FUNCTION_BLOCK fb_manual
VAR_INPUT
END_VAR
VAR_OUTPUT
END_VAR
VAR
	SFCInit : BOOL;
	fbi_paramInit: fb_paramInit;
	trn_paramInitDone: BOOL;

	fbi_jogController: fb_jogController;
	fbi_PTP : fb_PTP;
	fbi_operationElecylinder : fb_operationElecylinder;
	fbi_gm_operationElecylinder :fb_gm_operationElecylinder;
	fbi_oeprationChuck : fb_oeprationChuck;
	fbi_oeprationPush :fb_oeprationPush;
	fbi_operationEjector : fb_operationEjector;
	fbi_gm_operationEjector : fb_gm_operationEjector;
	fbi_recordingSystem : fb_recordingSystem;
	fbi_productGenerater : fb_productGenerator;
	fbi_gm_operationSV	: fb_gm_operationSV;
	var_i: INT;
	fbi_gm_setting: fb_gm_setting;
	fbi_gm_PTP: fb_gm_PTP;
	fbi_debugData: fb_debugData;
	var_cav_i: INT;
END_VAR

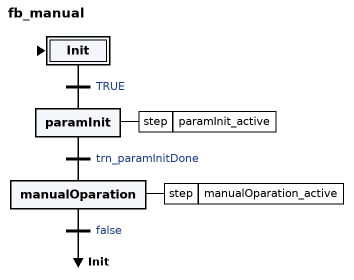
INITIAL_STEP Init:
END_STEP
TRANSITION FROM Init TO paramInit
    := TRUE;
END_TRANSITION
STEP paramInit:
    paramInit_active(N);  // step action
END_STEP
TRANSITION FROM paramInit TO manualOparation
    := trn_paramInitDone;
END_TRANSITION
STEP manualOparation:
    manualOparation_active(N);  // step action
END_STEP
TRANSITION FROM manualOparation TO Init
    := false;
END_TRANSITION

ACTION manualOparation_active:
IF manualOparation._x AND manualOparation.x = FALSE THEN
	THIS^.fbi_PTP();
	THIS^.fbi_PTP.p_init := TRUE;
	THIS^.fbi_operationElecylinder();
	THIS^.fbi_operationElecylinder.p_Init := TRUE;
	THIS^.fbi_gm_operationElecylinder();
	THIS^.fbi_gm_operationElecylinder.p_Init := TRUE;
	THIS^.fbi_oeprationChuck();
	THIS^.fbi_oeprationChuck.p_Init := TRUE;
	THIS^.fbi_oeprationPush();
	THIS^.fbi_oeprationPush.p_Init := TRUE;
	THIS^.fbi_operationEjector();
	THIS^.fbi_operationEjector.p_Init := TRUE;
	THIS^.fbi_gm_operationEjector();
	THIS^.fbi_gm_operationEjector.p_Init := TRUE;
	THIS^.fbi_gm_operationSV();
	THIS^.fbi_gm_operationSV.p_Init := TRUE;
	fbi_gm_PTP(in_flg_run := FALSE);
	//test mode
	fbi_debugData();
ELSIF manualOparation._x AND manualOparation.x THEN
	
//operation jog
	THIS^.fbi_jogController();
//PTP
	THIS^.fbi_PTP();
	THIS^.fbi_PTP.p_init := FALSE;
	fbi_gm_PTP(in_flg_run := TRUE);
//operation elecylinder
	THIS^.fbi_operationElecylinder();
	THIS^.fbi_operationElecylinder.p_Init := FALSE;
	THIS^.fbi_gm_operationElecylinder();
	THIS^.fbi_gm_operationElecylinder.p_Init := FALSE;
//operation chuck
	THIS^.fbi_oeprationChuck();
	THIS^.fbi_oeprationChuck.p_Init := FALSE;
	THIS^.fbi_gm_operationSV();
	THIS^.fbi_gm_operationSV.p_Init := FALSE;
//operation push
	THIS^.fbi_oeprationPush();
	THIS^.fbi_oeprationPush.p_Init := FALSE;
//operation ejector
	THIS^.fbi_operationEjector();
	THIS^.fbi_operationEjector.p_Init := FALSE;
	THIS^.fbi_gm_operationEjector();
	THIS^.fbi_gm_operationEjector.p_Init := FALSE;
//recording teach position
	THIS^.fbi_recordingSystem();
	fbi_gm_setting();
//new product generater
	THIS^.fbi_productGenerater();
//reset defective qty
	IF gvl_visu.flg_btn_clrDefectiveQty THEN
		FOR var_i := 1 TO 8 BY 1 DO
			gvl_auto.var_defectiveLens[var_i] := 0;
		END_FOR
	END_IF
//reset pocket qty
	IF gvl_visu.flg_btn_clrPockertQty THEN
		gvl_auto.flg_pocketCountCheck := false;
		FOR var_i := 1 TO 8 BY 1 DO
			gvl_auto.pocketNo[var_i] := 0;
		END_FOR
	END_IF
//reset gate length data
	IF gvl_visu.flg_btn_clrGateData THEN
		FOR var_i := 49 TO 0 BY -1 DO
			gvl_visu.var_gateLengthList[var_i] := 0;
			FOR var_cav_i := 1 TO 8 DO
				gvl_visu.var_gateLengthListCav[var_cav_i][var_i] := 0;
			END_FOR
		END_FOR
	END_IF
END_IF
//gate measurement run preset
	IF gvl_visu.flg_btn_gateMeasurementPreset THEN
		gvl_io.var_gateMeasurementPreset := 1;
	ELSE
		gvl_io.var_gateMeasurementPreset := 0;
	END_IF
END_ACTION

PROPERTY p_Init : bool
GET
p_init := THIS^.SFCInit;
END_GET
SET
THIS^.SFCInit := p_init;
END_SET
END_PROPERTY

ACTION paramInit_active:
fbi_paramInit(in_flg_run:= , out_flg_done=> );
IF paramInit._x AND paramInit.x = FALSE THEN
	trn_paramInitDone:= FALSE;
	fbi_paramInit.in_flg_run := FALSE;
ELSIF paramInit._x AND paramInit.x THEN
	fbi_paramInit.in_flg_run := TRUE;
	IF fbi_paramInit.out_flg_done THEN
		fbi_paramInit.in_flg_run := FALSE;
		trn_paramInitDone := TRUE;
	END_IF
END_IF
END_ACTION

END_FUNCTION_BLOCK

(* stored: Version 1.1.0.1, ProductVersion 3.1.4024.11
   POU fb_manual: Id {fa308f5f-6846-4dc5-b984-480947e3a377}, SpecialFunc None
   Action manualOparation_active: Id {534ca73a-2510-432a-a93c-ee45cc344769}
   Property p_Init: Id {39c8d22a-bdca-44cf-a8a7-432582d7bac9}
   Get Get: Id {da1a0b75-e1c2-4978-bdf2-430f760d6283}
   Set Set: Id {c2612c98-b1e9-46b0-bad3-9bb1dc581dc7}
   Action paramInit_active: Id {ad327194-c2b4-4821-8d34-dbf4ad8ec64c} *)
